{attribute 'qualified_only'}
VAR_GLOBAL
END_VAR

(* stored: Version 1.1.0.1, ProductVersion 3.1.4022.7
   GVL GVL_04_Auto_Step_Motor: Id {9df35170-f4f0-4200-842e-6c3e54748f27} *)
